SUBAPPLICATION SUBSCRIBE_R_TRIG (* Subscribed AX-Wert (per ID) auf steigende Flanke ueberwachen und als Event ausgeben *)
  (* Standard: 61499-2; Description: Copyright (c) 2026 HR Agrartechnik GmbH This program and the accompanying materials are made available under the terms of the Eclipse Public License 2.0 which is available at https://www.eclipse.org/legal/epl-2.0/ SPDX-License-Identifier: EPL-2.0 *)
  (* Version 2.0, 2026-09-11, Franz Höpfinger, HR Agrartechnik GmbH, Redundanten doppelten D_FF entfernt: vorher AX_SUBSCRIBE_1 (mit eigenem E_D_FF-Puffer) gefolgt von AX_R_TRIG (mit eigenem E_R_TRIG-Flankenspeicher) - 2 Speicher hintereinander fuer 1 Flankenerkennung. Jetzt direkt das rohe SUBSCRIBE_1 + E_R_TRIG verdrahtet (SUBSCRIBE_1.IND/RD_1 direkt in E_R_TRIG.EI/QI), nur noch 1 Speicherzustand. *)
  (* Version 1.0, 2026-08-26, Franz Höpfinger, HR Agrartechnik GmbH, initial API and implementation *)
  PACKAGE MyLib::sys;
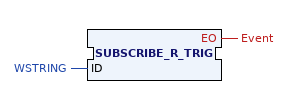
  EVENT_OUTPUT
    EO; (* Feuert bei steigender Flanke des subscribed AX-Werts *)
  END_EVENT
  VAR_INPUT
    ID : WSTRING; (* OPC-UA-Endpoint-Konstante (READ), z. B. Anlage_EIN_READ *)
  END_VAR
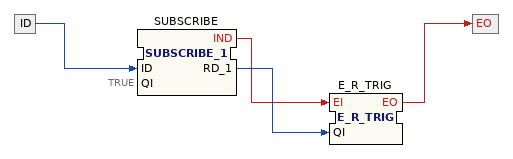
  FBS
    SUBSCRIBE : iec61499::net::SUBSCRIBE_1(QI := TRUE);
    E_R_TRIG : iec61499::events::E_R_TRIG;
  END_FBS
  EVENT_CONNECTIONS
    SUBSCRIBE.IND TO E_R_TRIG.EI;
    E_R_TRIG.EO TO EO;
  END_CONNECTIONS
  DATA_CONNECTIONS
    ID TO SUBSCRIBE.ID;
    SUBSCRIBE.RD_1 TO E_R_TRIG.QI;
  END_CONNECTIONS
END_SUBAPPLICATION
